INTERFACE I_LampCtrl

METHOD OFF : BOOL
END_METHOD

METHOD ON : BOOL
END_METHOD

PROPERTY State : STRING
GET
END_GET
END_PROPERTY

END_INTERFACE

(* stored: Version 1.1.0.1, ProductVersion 3.1.4024.6
   Itf I_LampCtrl: Id {aa66a24f-fc99-4589-ba32-3a83526bd01b}
   Method OFF: Id {6928b3c4-a764-4b4d-a0d3-428b9c9a2c5b}
   Method ON: Id {9642ddf5-d91c-422e-b5be-0c7f53d3ab3d}
   Property State: Id {8895653f-91e9-4f01-805e-7e753db19c5d}
   Get Get: Id {480ed50a-029a-4f43-981b-1d8b17b6d8f1} *)
